// TIA Portal V17 export
// export: Created 2025-03-05T08:03:28.9439356Z, ExportSetting WithDefaults, DisplayName Totally Integrated Automation Portal, DisplayVersion V17 Update 8, DisplayName TIA Portal Openness, DisplayVersion V17 Update 8, DisplayName TIA Portal Version Control Interface, DisplayVersion V17, DisplayName SINAMICS Startdrive Advanced, DisplayVersion V17 SP2, DisplayName SINAMICS Startdrive G110M, G120, G120C, G120D, G120P, G115D, DisplayVersion V17 SP2, DisplayName SINAMICS Startdrive G130, G150, S120, S150, SINAMICS MV, S210, DisplayVersion V17 SP2, DisplayName STEP 7 Professional, DisplayVersion V17 Update 8, DisplayName SINUMERIK ONE STEP 7 Toolbox, DisplayVersion V17 Update 12, DisplayName SINUMERIK 840D sl STEP 7 Toolbox, DisplayVersion V17 Update 12, DisplayName STEP 7 Safety, DisplayVersion V17 Update 6, DisplayName WinCC Advanced, DisplayVersion V17 Update 8
DATA_BLOCK "DB22503_PRESSURE_CONTROL_HOPPER_1_UNIT_01"   // DB22503
{ DB_Accessible_From_OPC_UA := 'FALSE' }
VERSION : 0.1
// stored: AutoNumber false, DBAccessibleFromOPCUA false, DBAccessibleFromWebserver true, InstanceOfName FB22500_PRESSURE_CONTROL_REGTONIC, InstanceOfType FB
"FB22500_PRESSURE_CONTROL_REGTONIC"
   // VAR_INPUT
   //    CONTROL_ON_DELAYED : Bool;
   //    PNEUMATIC_CONDITIONS : Bool;
   //    FEEDER_NOT_READY_FAULT : Bool;
   //    PRESSURIZE_VALVE_FEEDBACK : Bool;
   //    START_PROGRAM_REQUEST : Bool;
   //    START_MANUAL_REQUEST : Bool;
   //    START_SEMI_REQUEST : Bool;
   //    START_AUTO_REQUEST : Bool;
   //    STOP_PROGRAM_REQUEST : Bool;
   //    STOP_MANUAL_REQUEST : Bool;
   //    STOP_SEMI_REQUEST : Bool;
   //    STOP_AUTO_REQUEST : Bool;
   //    ACTUAL_PRESSURE : Real;
   //    PRESSURE_SETPOINT_AUTO : Real;
   // END_VAR
   // VAR_OUTPUT
   //    PRESSURE_CONTROL_VALUE : Int;
   //    SIMULTANEITY_ALARM : Bool;
   //    TIME_EXCEEDED_ALARM : Bool;
   //    SWITCH_ON_ALARM : Bool;
   //    SWITCH_OFF_ALARM : Bool;
   // END_VAR
   // VAR_IN_OUT
   //    DB_PID : PID_Compact;
   // END_VAR
   // VAR
   //    DATA_STANDARD : "GENERAL_DATA_START_STOP";
   //    START_STOP_HMI { S7_SetPoint := 'True'} : "HMI_DATA_START_STOP";
   //    INPUT_SETINGS : Struct
   //       UNIT_NUMBER : Int := 1;
   //       HOPPER_NUMBER : Int := 1;
   //    END_STRUCT;
   //    DATA_HMI : Struct
   //       PRESSURE_SETPOINT_VALUE : Real;
   //    END_STRUCT;
   //    ALARM_SETINGS : Struct
   //       TIMER_SIMULTANEITY : TON_TIME;
   //       TIMER_TIME_EXCEEDED { S7_SetPoint := 'True'} : TON_TIME;
   //    END_STRUCT;
   //    SETPOINT_PRESSURE : Real;
   //    CONTROL_PRESSURE_OUTPUT : Int;
   // END_VAR
BEGIN
END_DATA_BLOCK
